// TwinCAT 3 PLC project PLC
// ProgramVersion: 3.1.4024.0
// libraries:
//   Tc2_Standard, * (Beckhoff Automation GmbH)
//   Tc2_System, * (Beckhoff Automation GmbH)
//   Tc3_Module, * (Beckhoff Automation GmbH)
// project tree:
//   / PlcTask.TcTTO
//   POUs/ MAIN.TcPOU

CONFIGURATION PLC
    RESOURCE PLC ON TwinCAT3
        TASK PlcTask(INTERVAL := T#10ms, PRIORITY := 20);
        PROGRAM MAIN WITH PlcTask : MAIN;
    END_RESOURCE
END_CONFIGURATION

// ---- POUs/MAIN.TcPOU
PROGRAM MAIN
VAR
	bStart : BOOL := FALSE;
    bStop : BOOL := FALSE;
    bAlarm : BOOL := FALSE;
    iCounter : INT := 0;
    rTemperature : REAL := 20.0;
END_VAR


IF bStart THEN
    iCounter := iCounter + 1;
    rTemperature := rTemperature + 0.05;
END_IF

IF rTemperature > 30.0 THEN
    bAlarm := TRUE;
END_IF

IF bStop THEN
    bStart := FALSE;
    rTemperature := 20.0;
    bAlarm := FALSE;
    iCounter := 0;
END_IF

END_PROGRAM
